//{attribute 'hide_all_locals'}
FUNCTION_BLOCK PUBLIC DBAdaptor IMPLEMENTS ITF_DBAdaptor
VAR_INPUT
END_VAR
VAR_OUTPUT
END_VAR
VAR
	Database_Id	: UDINT := 0;
	sAmsNetId	: STRING(23) := '';
	tTimeOut	: TIME := T#1S;
	fbOpenConn	: FB_DBConnectionOpen;
	fbCloseConn	: FB_DBConnectionClose;
	fbAddConn	: FB_DBConnectionAdd;
	fbSqlDelete : FB_DBRecordDelete;
	fbSqlInsert : FB_DBRecordInsert_EX;
	fbSqlSelect : FB_DBRecordArraySelect;
	dbState 	: DB_State := DB_Idle;
	isOpened	: BOOL := FALSE;
END_VAR

;

{attribute 'object_name' := 'Close'}
METHOD PRIVATE Close : DB_FunctionResult
VAR_INPUT
END_VAR
IF isOpened THEN
	fbCloseConn(
		sNetID:= sAmsNetID, 
		hDBID:= Database_ID, 
		bExecute:= TRUE, 
		tTimeout:= tTimeOut );
	IF fbCloseConn.bBusy OR fbCloseConn.bError THEN 
		IF fbCloseConn.bError THEN 
			Close := DB_FunctionResult.DB_Error;
			fbCloseConn(
				sNetID:= sAmsNetId, 
				hDBID:= Database_ID, 
				bExecute:= FALSE, 
				tTimeout:= tTimeOut );
		END_IF
		IF fbCloseConn.bBusy THEN 
			Close := DB_FunctionResult.DB_Busy;
		END_IF
	ELSE
		fbCloseConn(
			sNetID:= sAmsNetId, 
			hDBID:= Database_ID, 
			bExecute:= FALSE, 
			tTimeout:= tTimeOut );
		isOpened := FALSE;
		Close := DB_FunctionResult.DB_Ok;
	END_IF
END_IF
END_METHOD

{attribute 'object_name' := 'SQL_Delete'}
METHOD SQL_Delete : DB_FunctionResult
VAR_INPUT
	SQL : STRING(255);
END_VAR
fbSqlDelete(
	sNetID:= sAmsNetId, 
	hDBID:= Database_Id, 
	pCmdAddr:= ADR(SQL), 
	cbCmdSize:= SIZEOF(SQL), 
	bExecute:= TRUE, 
	tTimeout:= tTimeOut );
IF fbSqlDelete.bBusy OR fbSqlDelete.bError THEN
	IF fbSqlDelete.bError THEN
		fbSqlDelete(
			sNetID:= sAmsNetId, 
			hDBID:= Database_Id, 
			pCmdAddr:= ADR(SQL), 
			cbCmdSize:= SIZEOF(SQL), 
			bExecute:= FALSE, 
			tTimeout:= tTimeOut );
		SQL_Delete := DB_FunctionResult.DB_Error;
	END_IF
	IF fbSqlDelete.bBusy THEN
		SQL_Delete := DB_FunctionResult.DB_Busy;
	END_IF
ELSE
	fbSqlDelete(
		sNetID:= sAmsNetId, 
		hDBID:= Database_Id, 
		pCmdAddr:= ADR(SQL), 
		cbCmdSize:= SIZEOF(SQL), 
		bExecute:= FALSE, 
		tTimeout:= tTimeOut );
	SQL_Delete := DB_FunctionResult.DB_Ok;
END_IF
END_METHOD

PROPERTY sNetID : STRING(23)
SET
sAmsNetId := sNetID;
END_SET
GET
sNetId := sAmsNetID;
END_GET
END_PROPERTY

{attribute 'object_name' := 'SQL_Insert'}
METHOD SQL_Insert : DB_FunctionResult
VAR_INPUT
	SQL : STRING(255);
END_VAR
fbSqlInsert(
	sNetID:= sAmsNetId, 
	hDBID:= Database_Id, 
	pCmdAddr:= ADR(SQL), 
	cbCmdSize:= SIZEOF(SQL), 
	bExecute:= TRUE, 
	tTimeout:= tTimeOut );
IF fbSqlInsert.bBusy OR fbSqlInsert.bError THEN
	IF fbSqlInsert.bError THEN
		fbSqlInsert(
			sNetID:= sAmsNetId, 
			hDBID:= Database_Id, 
			pCmdAddr:= ADR(SQL), 
			cbCmdSize:= SIZEOF(SQL), 
			bExecute:= FALSE, 
			tTimeout:= tTimeOut );
		SQL_Insert := DB_FunctionResult.DB_Error;
	END_IF
	IF fbSqlInsert.bBusy THEN
		SQL_Insert := DB_FunctionResult.DB_Busy;
	END_IF
ELSE
	fbSqlInsert(
		sNetID:= sAmsNetId, 
		hDBID:= Database_Id, 
		pCmdAddr:= ADR(SQL), 
		cbCmdSize:= SIZEOF(SQL), 
		bExecute:= FALSE, 
		tTimeout:= tTimeOut );
	SQL_Insert := DB_FunctionResult.DB_Ok;
END_IF
END_METHOD

{attribute 'object_name' := 'SQL_Select'}
METHOD SQL_Select : DB_FunctionResult
VAR_INPUT
	SQL 				: STRING(255);
	START_INDEX			: UDINT;
	ROWS				: UDINT;
	ROW_DATA_SIZE		: UDINT;
	ptr_ReceiveBuffer	: POINTER TO BYTE;
END_VAR
fbSqlSelect(
	sNetID:= sAmsNetId, 
	hDBID:= Database_ID, 
	pCmdAddr:= ADR(SQL), 
	cbCmdSize:= SIZEOF(SQL), 
	nStartIndex:= START_INDEX, 
	nRecordCount:= ROWS, 
	pDestAddr:= ptr_ReceiveBuffer, 
	cbRecordArraySize:= ROW_DATA_SIZE, 
	bExecute:= TRUE, 
	tTimeout:= tTimeOut );
IF fbSqlSelect.bBusy OR fbSqlSelect.bError THEN
	IF fbSqlSelect.bError THEN
		fbSqlSelect(
			sNetID:= sAmsNetId, 
			hDBID:= Database_ID, 
			pCmdAddr:= ADR(SQL), 
			cbCmdSize:= SIZEOF(SQL), 
			nStartIndex:= START_INDEX, 
			nRecordCount:= ROWS, 
			pDestAddr:= ptr_ReceiveBuffer, 
			cbRecordArraySize:= ROW_DATA_SIZE, 
			bExecute:= TRUE, 
			tTimeout:= tTimeOut );
		SQL_Select := DB_FunctionResult.DB_Error;
	END_IF
	IF fbSqlSelect.bBusy THEN
		SQL_Select := DB_FunctionResult.DB_Busy;
	END_IF
ELSE
	fbSqlSelect(
		sNetID:= sAmsNetId, 
		hDBID:= Database_ID, 
		pCmdAddr:= ADR(SQL), 
		cbCmdSize:= SIZEOF(SQL), 
		nStartIndex:= START_INDEX, 
		nRecordCount:= ROWS, 
		pDestAddr:= ptr_ReceiveBuffer, 
		cbRecordArraySize:= ROW_DATA_SIZE, 
		bExecute:= FALSE, 
		tTimeout:= tTimeOut );
	SQL_Select := DB_FunctionResult.DB_Ok;
END_IF
END_METHOD

{attribute 'object_name' := 'Open'}
METHOD PRIVATE Open : DB_FunctionResult
VAR_INPUT
END_VAR
IF NOT isOpened THEN
	fbOpenConn(
		sNetID:= sAmsNetId, 
		hDBID:= Database_ID, 
		bExecute:= TRUE, 
		tTimeout:= tTimeOut );
	IF fbOpenConn.bBusy OR fbOpenConn.bError THEN 
		IF fbOpenConn.bError THEN 
			Open := DB_FunctionResult.DB_Error;
			fbOpenConn(
				sNetID:= sAmsNetId, 
				hDBID:= Database_ID, 
				bExecute:= FALSE, 
				tTimeout:= tTimeOut );
		END_IF
		IF fbOpenConn.bBusy THEN 
			Open := DB_FunctionResult.DB_Busy;
		END_IF
		
	ELSE
		fbOpenConn(
			sNetID:= sAmsNetId, 
			hDBID:= Database_ID, 
			bExecute:= FALSE, 
			tTimeout:= tTimeOut );
		isOpened := TRUE;
		Open := DB_FunctionResult.DB_Ok;
	END_IF
END_IF
END_METHOD

PROPERTY udiDatabase_ID : UDINT
SET
Database_ID := udiDatabase_Id;
END_SET
GET
udiDatabase_ID := Database_Id;
END_GET
END_PROPERTY

PROPERTY TimeOut : TIME
GET
TimeOut := tTimeOut;
END_GET
SET
tTimeOut := TimeOut;
END_SET
END_PROPERTY

END_FUNCTION_BLOCK

(* stored: Version 1.1.0.1, ProductVersion 3.1.0.36
   POU DBAdaptor: Id {abccab33-d3de-45b2-a197-271df6c757eb}, SpecialFunc None
   Method Close: Id {090301b5-d7a0-4c7e-83a9-c565563887ff}
   Method SQL_Delete: Id {14ba833c-692c-4c6b-bf26-b30e6177eab6}
   Property sNetID: Id {4cefc892-7388-4919-a6ab-42003f7a4774}
   Set Set: Id {9106b61e-84d0-44b0-bbef-1a3f3f8612d6}
   Get Get: Id {f4a37a04-4438-4060-96b3-e00de1762898}
   Method SQL_Insert: Id {813d7971-78c7-4d45-8f56-becb63644dad}
   Method SQL_Select: Id {878a5881-e6d5-4326-bd4d-c9c7cade3cd3}
   Method Open: Id {98cf4f32-e65d-4442-aa7e-5703dadb3f78}
   Property udiDatabase_ID: Id {c69aa44a-16c2-47d9-87cb-f0a1f1744985}
   Set Set: Id {6dbb0e79-b957-44b0-94f0-601aaa3e237a}
   Get Get: Id {f5b7895b-2f3f-4351-bfc4-a87831dd3a83}
   Property TimeOut: Id {e714d72f-15b2-42b7-bd8d-0287408d9a43}
   Get Get: Id {0aa313e0-09b3-4dfd-8325-becba9fb2057}
   Set Set: Id {4911bcf8-c03d-4056-a48b-b3ec1b70e513} *)
